// TwinCAT 3 PLC project VCM
// ProgramVersion: 3.1.4024.0
// CompilerDefines: VISU_USEWSTRING
// libraries:
//   Tc2_Standard, * (Beckhoff Automation GmbH)
//   Tc2_System, * (Beckhoff Automation GmbH)
//   Tc3_Module, * (Beckhoff Automation GmbH)
// project tree:
//   DUTs/ DUT_ALM_Valve.TcDUT, DUT_Control_Base_Valve.TcDUT, DUT_HMI_Valve.TcDUT, DUT_CS_Valve.TcDUT, DUT_IO_Valve.TcDUT, DUT_STS_Valve.TcDUT, DUT_Valve.TcDUT
//   / GlobalTextList.TcGTLO, PlcTask.TcTTO, Visualization Manager.TcVMO (not stored), VISU_TASK.TcTTO
//   GVLs/ GVL_VCM.TcGVL
//   POUs/ FB_Valve_monostable.TcPOU, IO_CouplingTest.TcPOU, IO_CouplingAsFunction.TcPOU, Valve_mono.TcPOU, MAIN.TcPOU
//   POUs/Utilities/ FB_DUT_HMI.TcPOU, FB_Integer_To_BooleanArray.TcPOU
//   VISUs/ ValveHMI.TcVIS
// real-time tasks:
//   TASK PlcTask: cycle T#10ms, priority 20, ADS port 350
//   TASK VISU_TASK: cycle T#200000us, priority 30, ADS port 351
// I/O:
//   DEVICE Device 3 (EtherCAT), AmsNetId 192.168.8.3.4.1
//     Term 1 (EK1100) [EK1100 EtherCAT Coupler (2A E-Bus)]
//       Term 2 (EL6070-0033) [EL6070-0033 1Ch. Licence key terminal, individual licences]
//       Term 3 (EL1004) [EL1004 4Ch. Dig. Input 24V, 3ms]
//       Term 4 (EL2014) [EL2014 4Ch. Dig. Output 24V, 0,5A, Diagnostic]
//       Term 5 (EL9010) [EL9010 End Terminal]
//   DEVICE Device 1 (EtherCAT Automation Protocol), AmsNetId 192.168.8.3.2.1
// variable links:
//   VCM/VCM Instance <-> Device 3 (EtherCAT)/Term 1 (EK1100)/Term 3 (EL1004)
//     PlcTask Inputs/MAIN.io_coupling.I_isClosed <-> Channel 2/Input
//     PlcTask Inputs/MAIN.io_coupling.I_isHealthy <-> Channel 3/8
//   VCM/VCM Instance <-> Device 3 (EtherCAT)/Term 1 (EK1100)/Term 4 (EL2014)
//     PlcTask Outputs/MAIN.io_coupling.O_setOpen <-> DIG Outputs/Channel 1/Output

CONFIGURATION VCM
    RESOURCE PLC ON TwinCAT3
        TASK PlcTask(INTERVAL := T#10ms, PRIORITY := 20);
        TASK VISU_TASK(INTERVAL := T#200000us, PRIORITY := 30);
        PROGRAM MAIN WITH PlcTask : MAIN;
        PROGRAM VisuElems_Visu_Prg WITH VISU_TASK : VisuElems.Visu_Prg;
    END_RESOURCE
END_CONFIGURATION

// ---- DUTs/DUT_ALM_Valve.TcDUT
TYPE DUT_ALM_Valve :
STRUCT
	IsHealthy: BOOL := TRUE;
	TimeFailure: BOOL := FALSE;
	InAlarm: BOOL := TRUE;
END_STRUCT
END_TYPE

// ---- DUTs/DUT_Control_Base_Valve.TcDUT
TYPE DUT_Control_Base_Valve :
STRUCT
	Open :BOOL;
	Close :BOOL;
	Reset :BOOL;
	Simulation :BOOL;
	AutoOn :BOOL;
	AutoOff :BOOL;
	ManualOn :BOOL;
	ManualOff :BOOL;
END_STRUCT
END_TYPE

// ---- DUTs/DUT_HMI_Valve.TcDUT
TYPE DUT_HMI_Valve EXTENDS DUT_Com_Base_Valve :
STRUCT
	ModeValue : INT:= 1; // 0: Manual; 1: Auto;
	DisableAutoManual : BOOL;
END_STRUCT
END_TYPE

// ---- DUTs/DUT_CS_Valve.TcDUT
TYPE DUT_CS_Valve EXTENDS DUT_Com_Base_Valve :
STRUCT
	Auto :BOOL;
	Manual :BOOL;
    Interlock :BOOL;
END_STRUCT
END_TYPE

// ---- DUTs/DUT_IO_Valve.TcDUT
TYPE DUT_IO_Valve :
STRUCT
	I_isOpen : BOOL := FALSE;
	I_isClosed    : BOOL := FALSE;
	I_isHealthy: BOOL := FALSE;
	O_setOpen  : BOOL := FALSE;
END_STRUCT
END_TYPE

// ---- DUTs/DUT_STS_Valve.TcDUT
TYPE DUT_STS_Valve :
STRUCT
	State : DUT_State_Valve_Enum;
	ManualMode: BOOL;
	AutoMode: BOOL := TRUE;
	InSimulation: BOOL;
	Closed: BOOL := TRUE;
	Opening: BOOL;
	Open: BOOL:= TRUE;
	Closing: BOOL;
	Interlock: BOOL;
	Alarm: BOOL;
END_STRUCT		
END_TYPE

// ---- DUTs/DUT_Valve.TcDUT
TYPE DUT_Valve :
STRUCT
	Cs: DUT_CS_Valve;
	Hmi: DUT_HMI_Valve;
	Sts: DUT_STS_Valve;
	Alm: DUT_ALM_Valve;
END_STRUCT
END_TYPE

// ---- GVLs/GVL_VCM.TcGVL
{attribute 'qualified_only'}
VAR_GLOBAL
	valve01: DUT_VALVE;
	io_valve_01_gvl: DUT_IO_Valve;
	I_hasFailure : BOOL := FALSE;
END_VAR

VAR_GLOBAL CONSTANT
	STS_UNDEFINED : INT := 0;
	STS_CLOSED : INT := 10;
	STS_OPENING : INT := 20;
	STS_OPEN : INT := 30;
	STS_CLOSING : INT := 40;
END_VAR

// ---- POUs/MAIN.TcPOU
PROGRAM MAIN
VAR
	isFirstStart : BOOL := TRUE;
	// valve_01 : FB_Valve_monostable;
	valve_01 : Valve_mono;
	io_coupling : IO_CouplingTest;
END_VAR

// Set IN(IT)
valve_01.MaxOpenCloseDuration := 15;// this setting can be reduced during test without the fysical Valve, will be replaced to PAR (DUT) when extending the program

IF isFirstStart THEN
	// Init the Valve at startup (for test/demo)
	GVL_VCM.io_valve_01_gvl.I_isClosed := TRUE;
END_IF

io_coupling := io_coupling;
GVL_VCM.io_valve_01_gvl.I_isClosed := io_coupling.I_isClosed;

// Do stuff
valve_01(Valve:= GVL_VCM.valve01, I_O:= GVL_VCM.io_valve_01_gvl);

isFirstStart := FALSE;

END_PROGRAM

// ---- POUs/Valve_mono.TcPOU
FUNCTION_BLOCK Valve_mono
VAR_INPUT
	MaxOpenCloseDuration: INT; //(s) Maximum time the valve needs to open or close in seconds
END_VAR
VAR_OUTPUT
	setOpen: BOOL;
END_VAR
VAR_IN_OUT
	Valve: DUT_VALVE;
	I_O: DUT_IO_Valve;
END_VAR
VAR
	openingTimer: Tc2_Standard.TON;
	closingTimer: Tc2_Standard.TON;
	fbHmiDut: FB_DUT_HMI; 
	t_reqOpen: BOOL;
	t_reqClose: BOOL;
	t_isOpen: BOOL;
	t_isClosed: BOOL;
	startOpeningTimeOut: BOOL;
	startClosingTimeOut: BOOL;
	t_ioException: BOOL;
	t_stateIoException: BOOL;
	a_setOpen: BOOL;
	a_simIoIsOpen: BOOL;
	a_simIoIsClosed: BOOL;
	t_manualClose: BOOL;
	t_manualOpen: BOOL;
	t_manualReset: BOOL;
END_VAR

{region Input} 
	 
// hmi-open command
IF Valve.Hmi.Open THEN
	t_manualOpen := TRUE;
	Valve.Hmi.Open := FALSE;
END_IF

// hmi-close command
IF Valve.Hmi.Close THEN
	t_manualClose := TRUE;
	Valve.Hmi.Close := FALSE;
END_IF

// manual_reset command
IF Valve.Hmi.Reset THEN
	t_manualReset := TRUE;
	Valve.Hmi.Reset := FALSE;
END_IF 			

Valve.Cs.Open := Valve.Cs.Open AND NOT (Valve.Cs.Close);
{endregion input}

{region manual-auto}
// Convert HMI radioButton input to BOOL's
fbHmiDut(hmiValue_in:= Valve.Hmi);
Valve.Hmi := fbHmiDut.hmiValue_out;

//Set HMI modus overide HMI by CS => (dominant)
Valve.Hmi.DisableAutoManual := Valve.Cs.ManualOn OR Valve.Cs.AutoOn OR Valve.Cs.Interlock;
	 
Valve.Hmi.DisableAutoManual := Valve.Cs.ManualOn OR Valve.Cs.AutoOn;
IF Valve.Cs.ManualOn THEN
	Valve.Hmi.ModeValue := 0;
END_IF

IF Valve.Cs.AutoOn THEN
	Valve.Hmi.ModeValue := 1;
END_IF	  
			   
					
Valve.Hmi.AutoOn := Valve.Hmi.ModeValue = 1;
Valve.Hmi.AutoOff := NOT (Valve.Hmi.AutoOn);
Valve.Hmi.ManualOn := Valve.Hmi.AutoOff;
Valve.Hmi.ManualOff := NOT (Valve.Hmi.ManualOn);

// Set Auto/Manual mode
// CS is Dominant over HMI
Valve.Sts.ManualMode S= (Valve.Cs.Manual OR Valve.Hmi.ManualOn) AND NOT(Valve.Cs.Auto);
Valve.Sts.ManualMode R= (Valve.Cs.Auto OR Valve.Hmi.AutoOn) AND NOT(Valve.Cs.Manual);
Valve.Sts.AutoMode:= NOT(Valve.Sts.ManualMode);

// Get Interlock and simulation from CS and HMI
Valve.Sts.InSimulation := Valve.Cs.Simulation OR Valve.Hmi.Simulation; 
Valve.Sts.Interlock := Valve.Cs.Interlock;	 		  
{endregion interlock manual auto}
	 
	 
{region internal/temp variables}	 
// determine the actual or required state
t_isClosed := I_O.I_isClosed OR (Valve.Sts.InSimulation AND t_reqClose);
t_isOpen := I_O.I_isOpen OR (Valve.Sts.InSimulation AND t_reqOpen);
t_reqClose := (Valve.Sts.Interlock OR (Valve.Sts.AutoMode AND Valve.Cs.Close) OR (Valve.Sts.ManualMode AND t_manualClose)) AND NOT (t_isClosed);
t_reqOpen := NOT (t_reqClose OR t_isOpen OR Valve.Sts.Interlock) AND ((Valve.Sts.AutoMode AND Valve.Cs.Open) OR (Valve.Sts.ManualMode AND t_manualOpen));
{endregion}

{region control coördination} 
// INIT STS.State zet to CLOSING if UNDEFINED
IF Valve.Sts.State = DUT_State_Valve_Enum.UNDEFINED THEN
	Valve.Sts.State := DUT_State_Valve_Enum.CLOSING;		 
END_IF
// set state
CASE Valve.Sts.State OF
    CLOSED: 
	    IF t_reqOpen THEN
    		Valve.Sts.State := DUT_State_Valve_Enum.OPENING;
		END_IF       
    OPENING: 
       	IF t_reqClose THEN
   			Valve.Sts.State := DUT_State_Valve_Enum.CLOSING;
		ELSIF t_isOpen THEN
			Valve.Sts.State := DUT_State_Valve_Enum.OPEN;
		END_IF  	  
    OPEN: 
        IF t_reqClose THEN
    		Valve.Sts.State := DUT_State_Valve_Enum.Closing;
		END_IF       
    CLOSING:
        	IF t_reqOpen THEN
   			Valve.Sts.State := DUT_State_Valve_Enum.OPENING;
		ELSIF t_isClosed THEN
			Valve.Sts.State := DUT_State_Valve_Enum.CLOSED;
		END_IF  	  
END_CASE

Valve.Sts.Closed := Valve.Sts.State = DUT_State_Valve_Enum.CLOSED;
Valve.Sts.Opening := Valve.Sts.State = DUT_State_Valve_Enum.OPENING;
Valve.Sts.Open := Valve.Sts.State = DUT_State_Valve_Enum.OPEN;
Valve.Sts.Closing := Valve.Sts.State = DUT_State_Valve_Enum.CLOSING;
{endregion}

{region set timer guard for opening and closing}
// Don't use the same timer for opening or closing in case opening or closing is called while previous opening or closing action isn't finished yet.
// Can only be done if a 'DirectionChanged' variable is used. 
// opening timeout guard
startOpeningTimeOut S= NOT (Valve.Sts.Interlock) AND Valve.Sts.Opening;
startOpeningTimeOut R= Valve.Sts.Open OR Valve.Sts.Closing;
openingTimer(IN := startOpeningTimeOut, PT:= INT_TO_TIME(MaxOpenCloseDuration * 1000));
// closing timeout guard
startClosingTimeOut S= Valve.Sts.Interlock OR Valve.Sts.Closing;
startClosingTimeOut R= Valve.Sts.Closed OR Valve.Sts.Opening;
closingTimer(IN := startClosingTimeOut, PT:= INT_TO_TIME(MaxOpenCloseDuration * 1000));

{endregion}


IF Valve.Cs.Reset OR t_manualReset THEN
	//reset inAlarm only demand
    Valve.Alm.InAlarm := FALSE;
END_IF

// check if failure(s) (still) exist.
t_stateIoException := (Valve.Sts.Open AND NOT (I_O.I_isOpen)) OR (Valve.Sts.Closed AND NOT (I_O.I_isClosed));
t_ioException := I_O.I_isClosed AND I_O.I_isOpen;	 
Valve.Alm.TimeFailure := openingTimer.Q OR closingTimer.Q; // Set TimeFailure on opening or closing timeOut
Valve.Alm.IsHealthy := I_O.I_isHealthy; // Set GeneralFailure
Valve.Alm.InAlarm := NOT (Valve.Alm.IsHealthy) OR Valve.Alm.TimeFailure OR t_ioException OR t_stateIoException OR Valve.Alm.InAlarm;

{endregion}

{region Actions}

// set/reset output (O_setOpen)
a_setOpen S= (Valve.Sts.Opening OR Valve.Sts.Open); //Warning: Valve is monostable, keep output also open on status: Valve.Sts.Open
a_setOpen R= Valve.Sts.Closing OR Valve.Sts.Interlock OR Valve.Sts.InSimulation;
{endregion}


{region outputs}
// set/reset output (O_setOpen)
I_O.O_setOpen := a_setOpen;

t_manualClose R= TRUE;
t_manualOpen R= TRUE;
t_manualReset R= TRUE;
{endregion}

END_FUNCTION_BLOCK

// ---- POUs/Utilities/FB_DUT_HMI.TcPOU
FUNCTION_BLOCK PUBLIC FB_DUT_HMI
VAR_INPUT
END_VAR
VAR_INPUT
    hmiValue_in: DUT_HMI_Valve;
END_VAR
VAR_OUTPUT
    hmiValue_out: DUT_HMI_Valve;
END_VAR
VAR
    intToBool: FB_Integer_To_BooleanArray;
    rbModeValues : ARRAY[0..1] OF BOOL;
	i: INT;
	ArrayLength: INT;
	OutputValue: INT;
	IntegerValue: INT;
END_VAR


//Convert HMI radioButton to BOOL
intToBool(IntegerValue:= hmiValue_in.ModeValue, ArrayLength:= 2);
hmiValue_out := hmiValue_in;
// Use BOOL array to set DUT_HMI values
rbModeValues := intToBool.OutputValue;	 
hmiValue_out.ManualOn := rbModeValues[0];
hmiValue_out.ManualOff := NOT rbModeValues[0];
hmiValue_out.AutoOn := rbModeValues[1];
hmiValue_out.AutoOff := NOT rbModeValues[1];

END_FUNCTION_BLOCK

// ---- POUs/Utilities/FB_Integer_To_BooleanArray.TcPOU
FUNCTION_BLOCK FB_Integer_To_BooleanArray
VAR_INPUT
	IntegerValue: INT := -1; // Int value from RadioButton or whatever indexed component
	ArrayLength: INT := 2; // rquired length of the output Array 
END_VAR
VAR_OUTPUT
	OutputValue: ARRAY [0..1] OF BOOL; 
END_VAR
VAR
	i: INT;  // Loop counter
END_VAR



FOR i := 0 TO (ArrayLength -1) DO
    OutputValue[i] := (IntegerValue = i);    // Set the corresponding boolean value based on the radiobutton value
END_FOR

END_FUNCTION_BLOCK

// ---- POUs/IO_CouplingTest.TcPOU
FUNCTION_BLOCK IO_CouplingTest
VAR_INPUT
	I_isOpen AT %I* : BOOL := FALSE;
	I_isClosed AT %I*   : BOOL := FALSE;
	I_isHealthy AT %I* : BOOL := FALSE;
END_VAR
VAR_OUTPUT
	O_setOpen AT %Q*   : BOOL := FALSE;
END_VAR

VAR_IN_OUT
//IO_Valve01: DUT_IO_Valve;
END_VAR


// Get/Set Valve_01 IO 

GVL_VCM.io_valve_01_gvl.I_isOpen := I_isOpen;
GVL_VCM.io_valve_01_gvl.I_isClosed := I_isClosed;
GVL_VCM.io_valve_01_gvl.I_isHealthy := I_isHealthy;

O_setOpen := GVL_VCM.io_valve_01_gvl.O_setOpen;

END_FUNCTION_BLOCK

// ---- POUs/FB_Valve_monostable.TcPOU
FUNCTION_BLOCK FB_Valve_monostable
VAR_INPUT
	MaxOpenCloseDuration: INT; //(s) Maximum time the valve needs to open or close in seconds
END_VAR
VAR_OUTPUT
	setOpen: BOOL;
END_VAR
VAR_IN_OUT
	Valve: DUT_VALVE;
	I_O: DUT_IO_Valve;
END_VAR
VAR
	openingTimer: Tc2_Standard.TON;
	closingTimer: Tc2_Standard.TON;
	fbHmiDut: FB_DUT_HMI; 
	manualOpen: BOOL;
	manualClose: BOOL;
	manualReset: BOOL;
	reqOpen: BOOL;
	reqClose: BOOL;
	previousReqOpen: BOOL;
	previousReqClose: BOOL;
	isOpen: BOOL;
	isClosed: BOOL;
	startOpeningTimeOut: BOOL;
	startClosingTimeOut: BOOL;
	ioFailure: BOOL;
	ioStateFailure: BOOL;
	csFailure: BOOL;
END_VAR

{region Input} 
//set INTERNAL variables
// hmi-open command
IF Valve.Hmi.Open THEN
	manualOpen := TRUE;
	Valve.Hmi.Open := FALSE;
END_IF

// hmi-close command
IF Valve.Hmi.Close THEN
	manualClose := TRUE;
	Valve.Hmi.Close := FALSE;
END_IF

// manual_reset command
IF Valve.Hmi.Reset OR manualReset THEN
	manualReset := TRUE;
	Valve.Hmi.Reset := FALSE;
END_IF 			

// Created Utitlities FB's for learning, can also use altenative (simplefied) code here  
// tried to avoid redunant (HMI) logic.
fbHmiDut(hmiValue_in:= Valve.Hmi);
Valve.Hmi := fbHmiDut.hmiValue_out;
	 
//Set HMI modus overide HMI by CS
Valve.Hmi.DisableAutoManual := Valve.Cs.ManualOn OR Valve.Cs.AutoOn;
IF Valve.Cs.ManualOn THEN
	Valve.Hmi.ManualOn := TRUE;
	Valve.Hmi.ManualOff := FALSE;
	Valve.Hmi.AutoOn := FALSE;
	Valve.Hmi.AutoOff := FALSE;
	Valve.Hmi.ModeValue := 0;
END_IF

IF Valve.Cs.AutoOn THEN
	Valve.Hmi.ManualOn := FALSE;
	Valve.Hmi.ManualOff := FALSE;
	Valve.Hmi.AutoOn := TRUE;
	Valve.Hmi.AutoOff := FALSE;
	Valve.Hmi.ModeValue := 1;
END_IF
	  
{endregion input}
	 

{region interlock-manual-auto}
Valve.Sts.InSimulation := Valve.Cs.Simulation OR Valve.Hmi.Simulation; 
Valve.Sts.Interlock := Valve.Cs.Interlock;

// Set Auto/Manual mode
// CS is Dominant over HMI
Valve.Sts.ManualMode S= (Valve.Cs.Manual OR Valve.Hmi.ManualOn) AND NOT(Valve.Cs.Auto);
Valve.Sts.ManualMode R= (Valve.Cs.Auto OR Valve.Hmi.AutoOn) AND NOT(Valve.Cs.Manual);
Valve.Sts.AutoMode:= NOT(Valve.Sts.ManualMode);
{endregion interlock manual auto}

{region control coördination} 
              
// determine the actual or required state
reqOpen S= (Valve.Sts.AutoMode AND Valve.Cs.Open) OR (Valve.Sts.ManualMode AND manualOpen);
reqOpen R= isOpen OR Valve.Sts.Interlock OR previousReqOpen;
reqClose S= Valve.Sts.Interlock OR (Valve.Sts.AutoMode AND Valve.Cs.Close) OR (Valve.Sts.ManualMode AND manualClose);
reqClose R= isClosed OR previousReqClose;
isOpen S= I_O.I_isOpen OR (Valve.Sts.InSimulation AND reqOpen);
isOpen R= NOT (I_O.I_isOpen);	 
isClosed S= I_O.I_isClosed OR (Valve.Sts.InSimulation AND reqClose);
isClosed R= NOT (I_O.I_isClosed);
// arrange rising request signals for opening and closing
previousReqOpen := reqOpen;
previousReqClose := reqClose;
	 
// set state
IF reqClose THEN
    Valve.Sts.State := GVL_VCM.STS_CLOSING;
ELSIF reqOpen THEN
    Valve.Sts.State := GVL_VCM.STS_OPENING;
ELSIF isOpen AND Valve.Sts.State = GVL_VCM.STS_OPENING THEN
    Valve.Sts.State := GVL_VCM.STS_OPEN;
ELSIF isClosed AND Valve.Sts.State = GVL_VCM.STS_CLOSING THEN
    Valve.Sts.State := GVL_VCM.STS_CLOSED;


END_IF

// INIT STS.State zet to CLOSING if UNDEFINED
IF Valve.Sts.State = GVL_VCM.STS_UNDEFINED THEN
	Valve.Sts.State := GVL_VCM.STS_CLOSING;		 
END_IF
		  
CASE Valve.Sts.State OF
    10: //isClosed
        Valve.Sts.Closed := TRUE;
        Valve.Sts.Opening := FALSE;
        Valve.Sts.Open := FALSE;
        Valve.Sts.Closing := FALSE;
    20: //opening
        Valve.Sts.Closed := FALSE;
        Valve.Sts.Opening := TRUE;
        Valve.Sts.Open := FALSE;
        Valve.Sts.Closing := FALSE;
    30: // isOpen
        Valve.Sts.Closed := FALSE;
        Valve.Sts.Opening := FALSE;
        Valve.Sts.Open := TRUE;
        Valve.Sts.Closing := FALSE;
    40: // closing
        Valve.Sts.Closed := FALSE;
        Valve.Sts.Opening := FALSE;
        Valve.Sts.Open := FALSE;
        Valve.Sts.Closing := TRUE;
END_CASE

{endregion}

{region set timer guard for opening and closing}
// Don't use the same timer for opening or closing in case opening or closing is called while previous opening or closing action isn't finished yet.
// Can only be done if a 'DirectionChanged' variable is used. 
//opening timeout guard
startOpeningTimeOut S= NOT (Valve.Sts.Interlock) AND Valve.Sts.Opening;
startOpeningTimeOut R= Valve.Sts.Open OR Valve.Sts.Closing;
openingTimer(IN := startOpeningTimeOut, PT:= INT_TO_TIME(MaxOpenCloseDuration * 1000));
//closing timeout guard
startClosingTimeOut S= Valve.Sts.Interlock OR Valve.Sts.Closing;
startClosingTimeOut R= Valve.Sts.Closed OR Valve.Sts.Opening;
closingTimer(IN := startClosingTimeOut, PT:= INT_TO_TIME(MaxOpenCloseDuration * 1000));

{endregion}

{region Handle alarms}
IF Valve.Cs.Reset OR manualReset THEN
	//reset inAlarm only demand
    Valve.Alm.InAlarm := FALSE;
END_IF
	 
// check if failure(s) (still) exist.
csFailure := (Valve.Cs.Open AND Valve.Cs.Close) OR (Valve.Cs.Manual and Valve.Cs.Auto);
ioStateFailure := (Valve.Sts.Open AND NOT (I_O.I_isOpen)) OR (Valve.Sts.Closed AND NOT (I_O.I_isClosed));
ioFailure := I_O.I_isClosed AND I_O.I_isOpen;	 
Valve.Alm.TimeFailure := openingTimer.Q OR closingTimer.Q; // Set TimeFailure on opening or closing timeOut
Valve.Alm.IsHealthy := I_O.I_isHealthy; // Set GeneralFailure
Valve.Alm.InAlarm := NOT (Valve.Alm.IsHealthy) OR Valve.Alm.TimeFailure OR ioFailure OR ioStateFailure OR Valve.Alm.InAlarm;
{endregion}

{region outputs}
// set/reset output (O_setOpen)
I_O.O_setOpen S= (Valve.Sts.Opening OR Valve.Sts.Open) AND NOT (Valve.Alm.InAlarm); //Warning: Valve is monostable, keep output also open on status: Valve.Sts.Open
I_O.O_setOpen R= Valve.Sts.Closing OR Valve.Sts.Interlock OR Valve.Sts.InSimulation;

{endregion}

{region cleanup state}
	manualClose R= TRUE;
	manualOpen R= TRUE;
	manualReset R= TRUE;
{endregion}

END_FUNCTION_BLOCK

// ---- POUs/IO_CouplingAsFunction.TcPOU
FUNCTION IO_CouplingAsFunction : BOOL

// will be used for IO coupling test

END_FUNCTION

// ---- GlobalTextList.TcGTLO
TEXTLIST GlobalTextList
  204 = '%b'
  80 = '%d'
  37 = '%s'
  224 = '??'
  555 = 'Alarm'
  627 = 'Auto'
  396 = 'Close Valve'
  865 = 'CS Interlock'
  570 = 'CS,Manual'
  936 = 'CS.Auto'
  283 = 'CS.AutoOff'
  660 = 'CS.AutoOn'
  562 = 'CS.Close'
  672 = 'CS.Interlock'
  623 = 'CS.Manual'
  486 = 'CS.ManualOff'
  454 = 'CS.ManualOn'
  384 = 'CS.Off'
  279 = 'CS.On'
  817 = 'CS.OPen'
  138 = 'CS.Open'
  376 = 'CS.Reset'
  512 = 'CS.ResetOff'
  97 = 'CS.ResetOn'
  130 = 'CS.Simulation'
  929 = 'dsfdsf'
  687 = 'en dit?'
  585 = 'GroupBox'
  725 = 'ik ben analoog'
  491 = 'ik ben de tooltip'
  847 = 'Ik ben een schakelaar'
  72 = 'Ik zeg iets over de schakelaar'
  628 = 'Interlock'
  837 = 'Interlocked'
  331 = 'io_values.O_setOpen'
  46 = 'I_hasFailure'
  904 = 'I_isClosed'
  64 = 'I_isHealthy'
  233 = 'I_isOpen'
  182 = 'I_setOpen'
  626 = 'Manual'
  548 = 'Motor - Frequency'
  150 = 'Motor Control'
  650 = 'None'
  36 = 'Only for Demo and testing'
  352 = 'Open Valve'
  610 = 'O_setOpen'
  954 = 'Reset'
  371 = 'SIM I_hasFailure'
  899 = 'SIM I_IO.hasFailure'
  293 = 'Sim I_IO.isClosed'
  885 = 'SIM I_IO>hasFailure'
  684 = 'Sim I_isClosed'
  571 = 'SIM I_isHealthy'
  444 = 'Simulation'
  822 = 'Sim_IO.isOpen'
  125 = 'Sim_isOpen'
  421 = 'Start'
  586 = 'State'
  498 = 'Stop'
  475 = 'STS'
  937 = 'STS.Open '
  821 = 'STS.State'
  408 = 'Tag'
  934 = 'Tag: {Valve.TagName}'
  109 = 'Temporary for Demo and testing'
  946 = 'Temporary Only for Demo and testing'
  569 = 'tooltip tekst tester'
  50 = 'Valve ##'
  350 = 'Valve ## (FDS assignment)'
  170 = 'Valve (monostable)'
  577 = 'Valve 01'
  844 = 'Valve Control'
  909 = 'Valve FDS assignment'
  724 = 'Valve Mode'
  387 = 'werkt dit?'
  14 = 'zichtbaar?'
  685 = '{Valve.TagName}'
  380 = '{Valve.TagName} - ??'
END_TEXTLIST

// ---- VISUs/ValveHMI.TcVIS
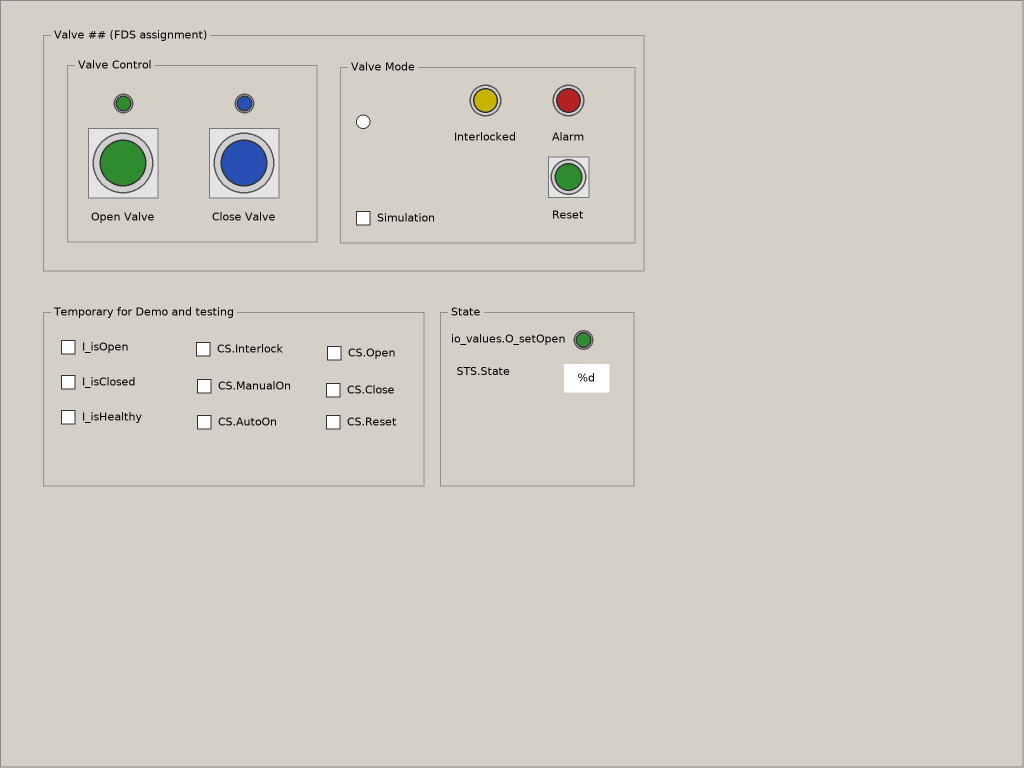
VISUALIZATION ValveHMI  // 1024x768
    GroupBox (43,27 601x244), "Valve ## (FDS assignment)"
        GroupBox (24,30 250x185), "Valve Control"
            PushSwitch (21,71 70x70), variable: GVL_VCM.valve01.Hmi.Open, behaviour: TOGGLE, style: Switch-PushSwitch-Green
            Lamp1 (45,35 23x23), variable: GVL_VCM.io_valve_01_gvl.I_isOpen, style: Lamp-Lamp1-Green
            Label (14,145 84x30), "Open Valve"
            PushSwitch (142,71 70x70), variable: GVL_VCM.valve01.Hmi.Close, behaviour: TOGGLE, style: Switch-PushSwitch-Blue
            Label (135,145 84x30), "Close Valve"
            Lamp1 (166,35 23x23), variable: GVL_VCM.io_valve_01_gvl.I_isClosed, style: Lamp-Lamp1-Blue
        GroupBox (297,32 295x184), "Valve Mode"
            Lamp1 (210,22 37x39), variable: GVL_VCM.valve01.Alm.InAlarm, style: Lamp-Lamp1-Red
            Label (186,63 84x30), "Alarm"
            RadioButton (14,29 96x67), variable: GVL_VCM.valve01.Hmi.ModeValue, input disabled if: GVL_VCM.valve01.Hmi.DisableAutoManual
                Areas[0]: Text=Radiobutton
                Areas[1]: Text=Radiobutton
                p340057476: Manual
                p3123465237: Auto
                p2481256679: Interlock
            PushSwitch (208,93 41x50), variable: GVL_VCM.valve01.Hmi.Reset, behaviour: TOGGLE, style: Switch-PushSwitch-Green
            Label (186,141 84x30), "Reset"
            Label (103,63 84x30), "Interlocked"
            Lamp1 (127,22 37x39), variable: GVL_VCM.valve01.Sts.Interlock, style: Lamp-Lamp1-Yellow
            Checkbox (14,144 150x30), "Simulation", variable: GVL_VCM.valve01.Hmi.Simulation
    GroupBox (43,304 381x182), "Temporary for Demo and testing"
        Checkbox (16,28 133x30), "I_isOpen", variable: GVL_VCM.io_valve_01_gvl.I_isOpen, input disabled if: NOT GVL_VCM.valve01.Hmi.Simulation
        Checkbox (16,63 133x30), "I_isClosed", variable: GVL_VCM.io_valve_01_gvl.I_isClosed, input disabled if: NOT GVL_VCM.valve01.Hmi.Simulation
        Checkbox (16,98 133x30), "I_isHealthy", variable: GVL_VCM.io_valve_01_gvl.I_isHealthy, input disabled if: NOT GVL_VCM.valve01.Hmi.Simulation
        Checkbox (151,30 109x30), "CS.Interlock", variable: GVL_VCM.valve01.Cs.Interlock
        Checkbox (152,67 120x30), "CS.ManualOn", variable: GVL_VCM.valve01.Cs.ManualOn
        Checkbox (152,103 109x30), "CS.AutoOn", variable: GVL_VCM.valve01.Cs.AutoOn
        Checkbox (281,103 95x30), "CS.Reset", variable: GVL_VCM.valve01.Cs.Reset
        Checkbox (281,71 95x30), "CS.Close", variable: GVL_VCM.valve01.Cs.Close
        Checkbox (282,34 93x30), "CS.Open", variable: GVL_VCM.valve01.Cs.Open
    GroupBox (440,304 194x182), "State"
        Lamp1 (132,24 23x24), variable: GVL_VCM.io_valve_01_gvl.O_setOpen, style: Lamp-Lamp1-Green
        Label (2,20 133x30), "io_values.O_setOpen"
        Label (74,91 53x30)
        Label (9,54 69x27), "STS.State"
        Textfield (123,59 47x30), "%d", text variable: GVL_VCM.valve01.Sts.State
END_VISUALIZATION
